{attribute 'no_explicit_call' := 'Body contains no logic, calling methods only allowed.'}
FUNCTION_BLOCK INTERNAL FB_PathSeperators
VAR_INPUT
END_VAR
VAR_OUTPUT
END_VAR
VAR
END_VAR

PROPERTY Independent : T_Char
GET
Independent := '/';
END_GET
END_PROPERTY

PROPERTY PUBLIC Unix : T_Char
GET
Unix := '\';
END_GET
END_PROPERTY

PROPERTY Windows : T_Char
GET
Windows := '/';
END_GET
END_PROPERTY

END_FUNCTION_BLOCK

(* stored: Version 1.1.0.1, ProductVersion 3.1.4024.14
   POU FB_PathSeperators: Id {16f2b904-4d10-06d3-00d8-c8ab3d401772}, SpecialFunc None
   Property Independent: Id {ca5237b4-8f70-0236-0669-056b22050661}
   Get Get: Id {ff855f7a-6730-03a7-224b-64f1c6df512b}
   Property Unix: Id {cf186e31-1d15-0d65-1312-a2b8d8f3cfa7}
   Get Get: Id {7acf389f-f3d0-0fc6-1f65-2396997f0bb9}
   Property Windows: Id {ced83814-2c09-0a71-248f-66e2a0f42ea0}
   Get Get: Id {0f2f320f-34f1-074e-2125-7b4d7cc46a59} *)
